FUNCTION_BLOCK FB_PWM
VAR_INPUT
	dutyCycle: LREAL;
END_VAR
VAR_OUTPUT
	state:BOOL;
END_VAR
VAR
	pulseWidth:INT;
	hertz:LREAL;
	currentTimeStep:INT;
	FB_GETCURTASKINDEX:GETCURTASKINDEX;
END_VAR

// a simple PWM function
FB_GETCURTASKINDEX();
Hertz:= 1 / (UDINT_TO_LREAL(_TaskInfo[FB_GETCURTASKINDEX.index].CycleTime)/ 10_000_000) ; // function takes the cycle time of the system to calculate the hertz
pulseWidth:=LREAL_TO_INT( hertz*dutyCycle); // the value is onverted to in to get rid of the values after the dot
currentTimeStep:= currentTimeStep+1;


IF currentTimeStep <= pulseWidth THEN // time on
	state:=TRUE;
ELSIF currentTimeStep >= hertz THEN // when finished
	state:=FALSE;
	currentTimeStep:=0;
ELSE // time off
	state:=FALSE;
END_IF

END_FUNCTION_BLOCK

(* stored: Version 1.1.0.1, ProductVersion 3.1.4024.9
   POU FB_PWM: Id {97f2005f-88d7-4913-9e3e-876430c870ed}, SpecialFunc None *)
